// TIA Portal V17 export
// export: Created 2026-04-13T11:12:54.1135355Z, ExportSetting WithDefaults, DisplayName Totally Integrated Automation Portal, DisplayVersion V17 Update 4, DisplayName TIA Portal Openness, DisplayVersion V17 Update 4, DisplayName TIA Portal Version Control Interface, DisplayVersion V17, DisplayName SINAMICS Startdrive Advanced, DisplayVersion V17, DisplayName SINAMICS Startdrive G130, G150, S120, S150, SINAMICS MV, S210, DisplayVersion V17, DisplayName SINAMICS Startdrive G110M, G120, G120C, G120D, G120P, G115D, DisplayVersion V17, DisplayName STEP 7 Professional, DisplayVersion V17 Update 4, DisplayName STEP 7 Safety, DisplayVersion V17, DisplayName WinCC Professional, DisplayVersion V17 Update 4
TagTable "OUTCIP"
  OUTCIP_DD电导合格值 : Real  (PLC tag OUTCIP.DD电导合格值, HMI_连接_1, 1 s)
  OUTCIP_JX碱洗温度设定 : Real  (PLC tag OUTCIP.JX碱洗温度设定, HMI_连接_1, 1 s)
  OUTCIP_DD电导率当前值 : Real  (PLC tag OUTCIP.DD电导率当前值, HMI_连接_1, 1 s)
  OUTCIP_JX碱洗温度 : Real  (PLC tag OUTCIP.JX碱洗温度, HMI_连接_1, 1 s)
  OUTCIP_CIP压力 : Real  (PLC tag OUTCIP.CIP压力, HMI_连接_1, 1 s)
  OUTCIP_MZD自动清洗 : Bool  (PLC tag OUTCIP.MZD自动清洗, HMI_连接_1, 1 s)
  OUTCIP_MSD手动_纯水清洗 : Bool  (PLC tag OUTCIP.MSD手动_纯水清洗, HMI_连接_1, 1 s)
  OUTCIP_MSD手动_碱水清洗 : Bool  (PLC tag OUTCIP.MSD手动_碱水清洗, HMI_连接_1, 1 s)
  OUTCIP_MSD手动_溶剂清洗 : Bool  (PLC tag OUTCIP.MSD手动_溶剂清洗, HMI_连接_1, 1 s)
  OUTCIP_MSD手动_热水清洗 : Bool  (PLC tag OUTCIP.MSD手动_热水清洗, HMI_连接_1, 1 s)
  OUTCIP_MQX清洗重置 : Bool  (PLC tag OUTCIP.MQX清洗重置, HMI_连接_1, 1 s)
  OUTCIP_MCS纯水罐阀门 : Bool  (PLC tag OUTCIP.MCS纯水罐阀门, HMI_连接_1, 1 s)
  OUTCIP_MJS碱水罐阀门 : Bool  (PLC tag OUTCIP.MJS碱水罐阀门, HMI_连接_1, 1 s)
  OUTCIP_MZS注射水阀门 : Bool  (PLC tag OUTCIP.MZS注射水阀门, HMI_连接_1, 1 s)
  OUTCIP_MYK压空吹干阀 : Bool  (PLC tag OUTCIP.MYK压空吹干阀, HMI_连接_1, 1 s)
  OUTCIP_MD清洗失败 : Bool  (PLC tag OUTCIP.MD清洗失败, HMI_连接_1, 1 s)
  OUTCIP_MQX室外清洗辅助 : Bool  (PLC tag OUTCIP.MQX室外清洗辅助, HMI_连接_1, 1 s)
  OUTCIP_MZT主塔清洗头 : Bool  (PLC tag OUTCIP.MZT主塔清洗头, HMI_连接_1, 1 s)
  OUTCIP_MZT中途停止 : Bool  (PLC tag OUTCIP.MZT中途停止, HMI_连接_1, 1 s)
  OUTCIP_MXT心跳信号发送 : Bool  (PLC tag OUTCIP.MXT心跳信号发送, HMI_连接_1, 1 s)
  OUTCIP_MXT心跳信号接受 : Bool  (PLC tag OUTCIP.MXT心跳信号接受, HMI_连接_1, 1 s)
  OUTCIP_MXY泄压请求 : Bool  (PLC tag OUTCIP.MXY泄压请求, HMI_连接_1, 1 s)
  OUTCIP_MGS供水泵请求 : Bool  (PLC tag OUTCIP.MGS供水泵请求, HMI_连接_1, 1 s)
  OUTCIP_MCIP远程状态 : Bool  (PLC tag OUTCIP.MCIP远程状态, HMI_连接_1, 1 s)
  OUTCIP_QCS纯水罐阀门 : Bool  (PLC tag OUTCIP.QCS纯水罐阀门, HMI_连接_1, 1 s)
  OUTCIP_QJS碱水罐阀门 : Bool  (PLC tag OUTCIP.QJS碱水罐阀门, HMI_连接_1, 1 s)
  OUTCIP_QZS注射水罐阀门 : Bool  (PLC tag OUTCIP.QZS注射水罐阀门, HMI_连接_1, 1 s)
  OUTCIP_QYG压干阀门 : Bool  (PLC tag OUTCIP.QYG压干阀门, HMI_连接_1, 1 s)
  OUTCIP_QGS供水泵状态CIP : Bool  (PLC tag OUTCIP.QGS供水泵状态CIP, HMI_连接_1, 1 s)
  OUTCIP_QXY泄压阀门 : Bool  (PLC tag OUTCIP.QXY泄压阀门, HMI_连接_1, 1 s)
  OUTCIP_PS排水时间 : Real  (PLC tag OUTCIP.PS排水时间, HMI_连接_1, 1 s)
  OUTCIP_PS排水时间计时 : Real  (PLC tag OUTCIP.PS排水时间计时, HMI_连接_1, 1 s)
